FUNCTION Convert_LWORD_TO_DATE : Hresult
VAR_INPUT
	in : LWORD;
	out : REFERENCE TO DATE;
END_VAR
VAR
	converted : DATE;
END_VAR
VAR CONSTANT
	INCOMPATIBLE : HRESULT := 16#9811070E;
END_VAR

converted := LWORD_TO_DATE(in);

IF (DATE_TO_LWORD(converted) <> in) THEN
	Convert_LWORD_TO_DATE := INCOMPATIBLE;
	RETURN;
END_IF

out := converted;

END_FUNCTION

(* stored: Version 1.1.0.1, ProductVersion 3.1.4024.12
   POU Convert_LWORD_TO_DATE: Id {7f623151-ace3-4d09-be4a-49d84c7a56b4}, SpecialFunc None *)
